TYPE DUT_STATEVALUES :
STRUCT
	Dummy:			BOOL := TRUE;				(*Free to use = TRUE, busy to use =FALSE*)
	Value:			LREAL;						(*Value of the State*)
	Name:			STRING[80];						(*Name of the state*)
	Description:	STRING[80];				(*Description of the state*)
	Unit:			STRING[80];						(*Unit of the state ()*)
END_STRUCT
END_TYPE

(* stored: Version 1.1.0.1, ProductVersion 3.1.0.25
   DUT DUT_STATEVALUES: Id {e9f73f70-854d-4689-b005-917fef921044} *)
